PROGRAM P_SqlSelectRecipe
VAR_INPUT
	bRead : BOOL; //Execute command
END_VAR
VAR
	
	fbSq : FB_EasySql;
	sSql : STRING(1000);
	
	iGE : INT:=1; //Select value
	
	astData : ARRAY[0..9] OF ST_SelectRecipeStruct; //Data array for recieved data
	
	bDone : BOOL; //Command done
	bError : BOOL; //Command error
	sError : STRING(255);
	
	udiNoOfRecords : UDINT; //Numbers of returned recoreds
	
END_VAR

//Select data from database
sSql := 'SELECT * from tpr_db.recipe WHERE recipe_id =¤1¤';

F_Replace(pString:= ADR(sSql), cbStringLen:= SIZEOF(sSql), sSearch:= '¤1¤', sReplace:= TO_STRING(PROGRAM_DATA.usiRecipe)); //Replace placeholder

fbSq(
	bExecute:= bRead, 
	wDBID:= 1, 
	pSql:= ADR(sSql), 
	cbSql:= SIZEOF(sSql), 
	pData:= ADR(astData), 
	cbData:= SIZEOF(astData), 
	udiMaxOfRecord:= 3, //Max number of recieved records
	udiNoOfRecords=> udiNoOfRecords, 
	bDone=> bDone, 
	bBusy=> , 
	bError=> bError, 
	sError=> sError
);

END_PROGRAM

(* stored: Version 1.1.0.1, ProductVersion 3.1.4024.4
   POU P_SqlSelectRecipe: Id {168a33c5-356e-4e3d-86f3-969421b345a2}, SpecialFunc None *)
